// TIA Portal project "Proyecto 2" (V17)

(* hardware
DEVICE "S7-1500/ET200MP station_1"  S7-1500 station
   slot 0: "Rail_0"  Rack  6ES7 590-1***0-0AA0
   slot 1: "PLC_1"  CPU 1515-2 PN  6ES7 515-2AM02-0AB0  V2.9
      slot 3: "CPU display_1"  6ES7591-1BA00-0AA0
      slot 32768: "PROFINET interface_1"  X1
         slot 32769: "Port_1"  X1 P1
         slot 32770: "Port_2"  X1 P2
      slot 33024: "PROFINET interface_2"  X2
         slot 33025: "Port_1"  X2 P1
      slot 34817: "Virtual CP interface port_1"  Virtual CP interface port  Virtual CP interface port
   slot 2: "AI 8xU/I/RTD/TC ST_1"  AI 8xU/I/RTD/TC ST  6ES7 531-7KF00-0AB0  V2.0
   slot 3: "AI 8xU/I/RTD/TC ST_2"  AI 8xU/I/RTD/TC ST  6ES7 531-7KF00-0AB0  V2.0
   slot 4: "AI 8xU/I/RTD/TC ST_3"  AI 8xU/I/RTD/TC ST  6ES7 531-7KF00-0AB0  V2.0
   slot 5: "AI 8xU/I/RTD/TC ST_4"  AI 8xU/I/RTD/TC ST  6ES7 531-7KF00-0AB0  V2.0
   slot 6: "DI 16x24VDC BA_1"  DI 16x24VDC BA  6ES7 521-1BH10-0AA0  V1.0
*)

// ===== PLC "PLC_1"  CPU 1515-2 PN =====

VAR_GLOBAL   // PLC tag table "Default tag table"
   "Pulsador Marcha" AT %I0.0 : Bool;
   "Pulsador Paro" AT %I0.1 : Bool;
   "Sensor A" AT %I0.2 : Bool;
   "Sensor B" AT %I0.3 : Bool;
   "Pulsador Led Marcha" AT %Q0.0 : Bool;
   "Pulsador Led Paro" AT %Q0.1 : Bool;
   "Led Marcha" AT %Q0.2 : Bool;
   "Led Paro" AT %Q0.3 : Bool;
   "Entry Conveyor" AT %Q0.4 : Bool;
   "Conveyor" AT %Q0.5 : Bool;
   "Permiso Marcha" AT %M0.0 : Bool;
   "Bloqueo" AT %M0.1 : Bool;
END_VAR

FUNCTION "MHJ-PLC-Lab-Function-S71500" : Void   // FC9000, SCL
{ S7_Optimized_Access := 'TRUE' }
VERSION : 0.1
   VAR_TEMP
      Value : Byte;
      ForCounter : Int;
   END_VAR
   VAR CONSTANT
      Value_01_DW : DWord := 16#1223_5486;
      Value_02_DW : DWord := 16#A6C9_D1F5;
   END_VAR
BEGIN

   #Value:=PEEK(area := 16#82,
        dbNumber := 0,
        byteOffset := 511);
   #Value := #Value + 1;

   POKE(area := 16#82,
        dbNumber := 0,
        byteOffset := 511,
        value := #Value);

   POKE(area := 16#82,
        dbNumber := 0,
        byteOffset := 1016,
        value := #Value_01_DW);
   POKE(area := 16#82,
        dbNumber := 0,
        byteOffset := 1020,
        value := #Value_02_DW);

   FOR #ForCounter := 0 TO 63 DO
       #Value:=PEEK(area := 16#1,
            dbNumber := 0,
            byteOffset := #ForCounter);
       POKE(area := 16#81,
            dbNumber := 0,
            byteOffset := #ForCounter,
            value := #Value);
   END_FOR;
   #Value := PEEK(area := 16#1,
                  dbNumber := 0,
                  byteOffset := 512);
   POKE(area := 16#82,
        dbNumber := 0,
        byteOffset := 512,
        value := #Value);
END_FUNCTION

ORGANIZATION_BLOCK "Main"   // OB1, LAD, ProgramCycle
TITLE = "Main Program Sweep (Cycle)"
{ S7_Optimized_Access := 'TRUE' }
VERSION : 0.1
   VAR_INPUT
      Initial_Call : Bool;   // Initial call of this OB
      Remanence : Bool;   // =True, if remanent data are available
   END_VAR
BEGIN

REGION Network 1: Conexion Factory I/O
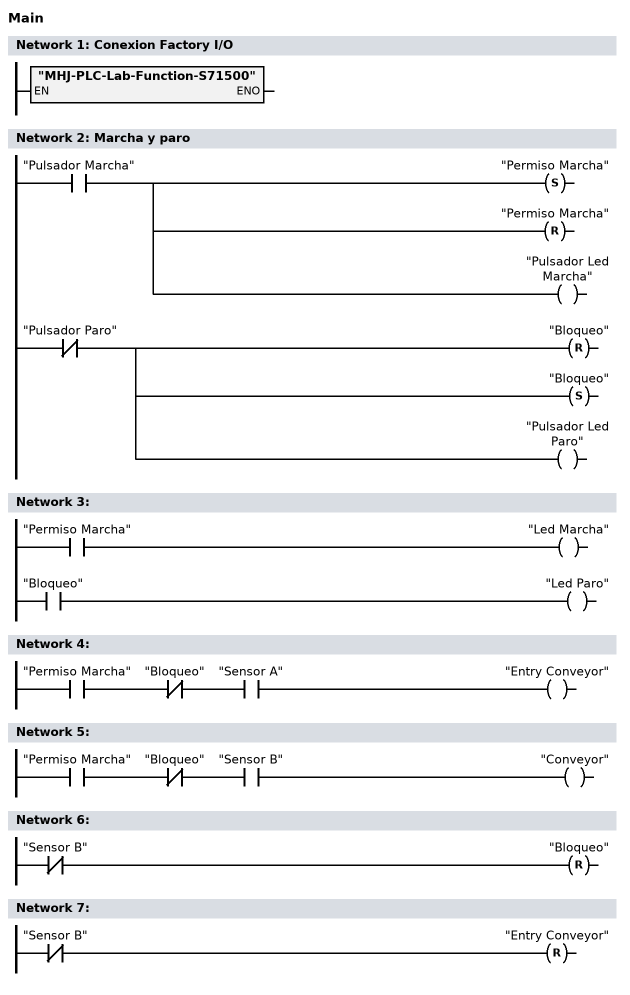
   RUNG wire#powerrail
      "MHJ-PLC-Lab-Function-S71500"()
   END_RUNG
   // the same network as SCL:
   "MHJ-PLC-Lab-Function-S71500"();
END_REGION

REGION Network 2: Marcha y paro
   RUNG wire#powerrail
      Contact( "Pulsador Marcha" )
      wire#w1
      S_Coil( "Permiso Marcha" )
   END_RUNG
   RUNG wire#w1
      R_Coil( "Permiso Marcha" )
   END_RUNG
   RUNG wire#w1
      Coil( "Pulsador Led Marcha" )
   END_RUNG
   RUNG wire#powerrail
      I_Contact( "Pulsador Paro" )
      wire#w2
      R_Coil( "Bloqueo" )
   END_RUNG
   RUNG wire#w2
      S_Coil( "Bloqueo" )
   END_RUNG
   RUNG wire#w2
      Coil( "Pulsador Led Paro" )
   END_RUNG
   // the same network as SCL:
   IF "Pulsador Marcha" THEN
       "Permiso Marcha" := TRUE;
       "Permiso Marcha" := FALSE;
   END_IF;
   "Pulsador Led Marcha" := "Pulsador Marcha";
   IF NOT "Pulsador Paro" THEN
       "Bloqueo" := FALSE;
       "Bloqueo" := TRUE;
   END_IF;
   "Pulsador Led Paro" := NOT "Pulsador Paro";
END_REGION

REGION Network 3
   RUNG wire#powerrail
      Contact( "Permiso Marcha" )
      Coil( "Led Marcha" )
   END_RUNG
   RUNG wire#powerrail
      Contact( "Bloqueo" )
      Coil( "Led Paro" )
   END_RUNG
   // the same network as SCL:
   "Led Marcha" := "Permiso Marcha";
   "Led Paro" := "Bloqueo";
END_REGION

REGION Network 4
   RUNG wire#powerrail
      Contact( "Permiso Marcha" )
      I_Contact( "Bloqueo" )
      Contact( "Sensor A" )
      Coil( "Entry Conveyor" )
   END_RUNG
   // the same network as SCL:
   "Entry Conveyor" := "Permiso Marcha" AND NOT "Bloqueo" AND "Sensor A";
END_REGION

REGION Network 5
   RUNG wire#powerrail
      Contact( "Permiso Marcha" )
      I_Contact( "Bloqueo" )
      Contact( "Sensor B" )
      Coil( "Conveyor" )
   END_RUNG
   // the same network as SCL:
   "Conveyor" := "Permiso Marcha" AND NOT "Bloqueo" AND "Sensor B";
END_REGION

REGION Network 6
   RUNG wire#powerrail
      I_Contact( "Sensor B" )
      R_Coil( "Bloqueo" )
   END_RUNG
   // the same network as SCL:
   IF NOT "Sensor B" THEN "Bloqueo" := FALSE; END_IF;
END_REGION

REGION Network 7
   RUNG wire#powerrail
      I_Contact( "Sensor B" )
      R_Coil( "Entry Conveyor" )
   END_RUNG
   // the same network as SCL:
   IF NOT "Sensor B" THEN "Entry Conveyor" := FALSE; END_IF;
END_REGION
END_ORGANIZATION_BLOCK